// TIA Portal V20 export
VAR_GLOBAL   // PLC tag table "CentralFunctions"
END_VAR
